// TwinCAT 3 PLC project Untitled1
// ProgramVersion: 3.1.4023.0
// libraries:
//   Tc2_Standard, * (Beckhoff Automation GmbH)
//   Tc2_System, * (Beckhoff Automation GmbH)
//   Tc3_Module, * (Beckhoff Automation GmbH)
// project tree:
//   / PlcTask.TcTTO
//   POUs/ FB_RPC.TcPOU, MAIN.TcPOU
// real-time tasks:
//   TASK PlcTask: cycle T#10ms, priority 20, ADS port 350

CONFIGURATION Untitled1
    RESOURCE PLC ON TwinCAT3
        TASK PlcTask(INTERVAL := T#10ms, PRIORITY := 20);
        PROGRAM MAIN WITH PlcTask : MAIN;
    END_RESOURCE
END_CONFIGURATION

// ---- POUs/MAIN.TcPOU
PROGRAM MAIN
VAR
	fb_rpc : FB_RPC;
END_VAR

END_PROGRAM

// ---- POUs/FB_RPC.TcPOU
FUNCTION_BLOCK FB_RPC
VAR_INPUT
END_VAR
VAR_OUTPUT
END_VAR
VAR
	m_cnt_add : UINT;
END_VAR

{attribute 'TcRpcEnable'}
METHOD M_Add : DINT
VAR_INPUT
	a : DINT;
	b : DINT;
END_VAR
m_cnt_add := m_cnt_add +1;
M_Add := a + b;
END_METHOD

END_FUNCTION_BLOCK
